KUKA KRL program: fri_isir_default.src, fri_isir_default.dat

--- fri_isir_default.src ---
&ACCESS RVP
&REL 1
&PARAM TEMPLATE = C:\KRC\Roboter\Template\vorgabe
&PARAM EDITMASK = *
DEF run_fri_isir_default( )

; User Parameters

fri_rate_ms = 1
tool_number = 5
base_number = 0

; Go To Zero ;
;PTP HOME
; Go To start Pos ;
;PTP {a1 90,a2 90,a3 -90,a4 0,a5 90,a6 0,e1 0}

;FOLD FRI ISIR Control ()
fri_isir(fri_rate_ms,tool_number,base_number)
;ENDFOLD

END

--- fri_isir_default.dat ---
&ACCESS RVP
&REL 1
&PARAM TEMPLATE = C:\KRC\Roboter\Template\vorgabe
&PARAM EDITMASK = *
DEFDAT run_fri_isir_default

;FOLD EXTERNAL DECLARATIONS;%{PE}%MKUKATPBASIS,%CEXT,%VCOMMON,%P
;FOLD BASISTECH EXT;%{PE}%MKUKATPBASIS,%CEXT,%VEXT,%P
EXT  BAS (BAS_COMMAND  :IN,REAL  :IN )



DECL INT fri_rate_ms
DECL INT tool_number
DECL INT base_number

EXT fri_isir(INT:IN,INT:IN,INT:IN )


;ENDFOLD (BASISTECH EXT)
;FOLD USER EXT;%{E}%MKUKATPUSER,%CEXT,%VEXT,%P
;Make here your modifications

;ENDFOLD (USER EXT)
;ENDFOLD (EXTERNAL DECLARATIONS)
ENDDAT
